// TIA Portal V17 export
// export: Created 2024-09-15T12:30:12.3257255Z, ExportSetting WithDefaults, DisplayName Totally Integrated Automation Portal, DisplayVersion V17, DisplayName TIA Portal Openness, DisplayVersion V17, DisplayName TIA Portal Version Control Interface, DisplayVersion V17, DisplayName STEP 7 Professional, DisplayVersion V17, DisplayName STEP 7 Safety, DisplayVersion V17, DisplayName WinCC Professional, DisplayVersion V17
DATA_BLOCK "SLD_Tracking_DB"   // DB52
VERSION : 0.1
// stored: AutoNumber true, DBAccessibleFromOPCUA true, DBAccessibleFromWebserver true, InstanceOfName SLD_Tracking, InstanceOfType FB
"SLD_Tracking"
   // VAR
   //    Location : String;
   // END_VAR
BEGIN
END_DATA_BLOCK
